(* CODESYS project CtaAppLeistungsreduktion_2.0.0.0.library
   Description: Leistungsreduktion Library der CTA
   Version: 2.0.0.0
   Title: CtaAppLeistungsreduktion
   Author: SIS
   DocFormat: reStructuredText
   LanguageModelAttribute: qualified-access-only
   Placeholder: CtaAppLeistungsreduktion
   DefaultNamespace: CtaAppLeistungsreduktion
   CompiledLibraryCompatibilityVersion: CODESYS V3.5 SP16 Patch 3
   Company: CTA

Project tree, tasks and I/O mapping:
  libraries: CtaSysConfig, 2.0.0.0 (CTA); CtaAppTime, 1.0.0.1 (CTA); CtaAppPid, 2.0.0.0 (CTA); Standard, 3.5.18.0 (System); VisuSymbols, 4.5.0.0 (System); CtaVisSymbols, 2.0.0.0 (CTA); CtaAppInfluxLog, 1.0.0.1 (CTA); VisuDialogs, * (System); CtaVisApps, 1.0.0.0 (CTA); CtaVisHelp, 1.0.0.0 (CTA); CtaVisUser, 1.0.0.0 (CTA)
  40 Visualizations/
    visualisation visLeistungsreduktion
    Powerreduction/
      Rectangles/
        visualisation visPowerReduktion4eck
        visualisation visPowerReduktion4eckCircuit
        visualisation visPowerReduktion4eckCircuitSingle
        visualisation visPowerReduktionSingle
      Combinations/
        visualisation visPrCircuit
        visualisation visPrCircuitSingle
      VisIcons/
        Circuits/
          SingleCompressor/
            visualisation visPowerReduktionKreisInOnly
            visualisation visPowerReduktionKreis
          DualCompressor/
            visualisation visPowerReduktionKreis2V
            visualisation visPowerReduktionKreis2VInOnly
        GeneralPowerreductions/
          visualisation visPrIn
          visualisation visPrInOut
          visualisation visPrOut
          visualisation visPrNoInOut
    Parameter/
      visualisation Parameter
    Dialogs/
      visualisation visLeistungsreduktionManager
      visualisation visLrZeile
  30 Program Organization Units/
    function block fbLeistungsReduktionManager [ST]
    function block fbLeistungsReduktion [ST]: actConfig, actTrendLog, actLeistungreduktion
  00000000-0000-0000-0000-000000000000|D:\CoDeSys\LibrariesV3\trunk\Intern\CAA\CAA Template\3.4.0.0 draft\Placeholder.xml
  00000000-0000-0000-0000-000000000000|D:\CoDeSys\LibrariesV3\trunk\Intern\CAA\CAA Template\3.2.0.3 draft\Prefix.pdf
  00000000-0000-0000-0000-000000000000|D:\CoDeSys\LibrariesV3\trunk\Intern\CAA\CAA Template\3.5.2.0 draft\Placeholder.xml
  20 Structs/
    data type scParameter
  50 Images/
  10 Documenation/
    global variables VersionHistory
    global variables readMe
  21 Interface/
  11 Library Parameter/
  12 Konstanten/
  60 Textlisten/
  13 Globale Variablen/
  text list GlobalTextList
*)

// 20 Structs/scParameter
TYPE scParameter :
    STRUCT
        fbxEn                         :   CtaSysConfig.fbBOOL;   // 1=Leistungsreduktion Überwachung aktivieren/deaktivieren
        fbtStartTime                  :   CtaSysConfig.fbTIME;   // Ton1= Sobald Verdichter/Anlage aktiv ist wird die Leistungsreduktion gemäss StartTime Einschaltverzögert
        fbtRunTime                    :   CtaSysConfig.fbTIME;   // Ton2= Sobald der Istwert den Sollwert überschreitet/unterschreitet wird die Leistungsreduktion minimum gemäss RunTime Einschaltverzögert unabhängig von Ton1
        fbrCounter                    :   CtaSysConfig.fbREAL;   // Soviel% wird in einer Sekunde angeglichen 0% zu PI Regler
        fbrSoll                       :   CtaSysConfig.fbREAL;   // Sollwert
        fbxEnTrendLog                 :   CtaSysConfig.fbBOOL;   // Trendlog Aktivieren       
    END_STRUCT
END_TYPE

// 10 Documenation/VersionHistory
(* 

.. image:: ../../Images/CTA_Logo.jpg
   :align: right
   :width: 15% 

**Vorlage**   


============ =========== =========== ============================================
**Date**     **Version** **Author**  **Change**
------------ ----------- ----------- --------------------------------------------
04.03.2021   0.0.0.0     SIS         Vorlage erstellt

============ =========== =========== ============================================


*)
VAR_GLOBAL
    stInfo : STRING:= '0.0.0.0, Vorlage, CTA';
END_VAR

// 10 Documenation/readMe
(*

**ReadMe**
 
|	**Empfehlung**
|
|	Die Bibliothek CtaAppLeistungredukton dient der reduktion der Leistung unter Berücksichtigung der definierten Parameter.
|	Instanzieren Sie den CtaAppLeistungredukton.fbLeistungsReduktion in ihrem Funktionsbaustein oder POU beispielsweise als fbLrx (x = Nr. der Leistungsreduktion)
|	Deklarieren Sie die Struktur Variable welche als Parameter und zur ansteuerung dienen wie im Code beispiel.
|  
| *Beispiel* 

+-----------------------+---------------------------------------------------------------------------------------------------------------------------------------------------------------------------------------------------------------------------------------------------------------------------------------------------------------------------------------------------------------------------------------------------------------------------------------+
| Beschreibung          |  Code                                                                                                                                                                                                                                                                                                                                                                                                                                 |
+=======================+=======================================================================================================================================================================================================================================================================================================================================================================================================================================+
| Pou oder SmFb         | .. code-block:: codesys                                                                                                                                                                                                                                                                                                                                                                                                               |
|                       |                                                                                                                                                                                                                                                                                                                                                                                                                                       |
|                       |	// Deklaration als VAR im POU oder dem selbsterstellten Funktionsbaustein                                                                                                                                                                                                                                                                                                                                                       	|
|                       |   VAR   																																																																																																								|
|						|	    (*Leistungsreduktionen*)																																																		 																																																|
|						|		fbLr1			: CtaAppLeistungredukton.fbLeistungsReduktion;                                                                                                                                                                                                                                                                                                                                                              	|
|						|																																																																																																										|
+-----------------------+---------------------------------------------------------------------------------------------------------------------------------------------------------------------------------------------------------------------------------------------------------------------------------------------------------------------------------------------------------------------------------------------------------------------------------------+
| Code für Init         | .. code-block:: codesys                                                                                                                                                                                                                                                                                                                                                                                                               |
|                       |   																																																																																																									|
| 						|	// Kopieren des nachfolgenden Codes in eine Action zur Initialisierung der Parameter. Zum Beispiel actConfig.																																																																														|
|                       |	{region " Stufenschaltung "}                                                                                                                                                                                                                                                                                                                                                                                                     	|
| 						|		(*Basis*)																																																																																																						|
|						|		fbLr1.scParameter.fbxEn               				(_wertInit :=	 FALSE														);		//P1 Leistungsreduktion aktiv / inaktiv																																																													|
|						|		fbLr1.scParameter.fbtStartTime						(_wertInit :=	 T#30s		, _minInit :=			, _maxInit :=			);		//P2 Einschaltverzögerung der Leistungsreduktion nach Start des Verdichters / der Analge																																																| 
|						|		fbLr1.scParameter.fbtRunTime						(_wertInit :=	 T#30s		, _minInit :=			, _maxInit :=			);		//P3 Einschaltverzögerung der Leistungsreduktion im Betrieb bei Unter- oder Überschreitung des Sollwertes																																												| 
|						|		fbLr1.scParameter.fbrCounter						(_wertInit :=		15		, _minInit :=			, _maxInit := 			);		//P4 Wert für Angleichung innert einer Sekunde																																																											| 
|						|		fbLr1.scParameter.fbrSoll							(_wertInit := 		30		, _minInit :=   		, _maxInit := 			);		//P5 Sollwert																																																																			|
|						|		fbLr1.scParameter.fbxEnTrendLog						(_wertInit := 	  TRUE														);		//P6 Aktivierung der Trendaufzeichnung 																																																													|
|						|	{endregion}                                                                                                                                                      																																																																	| 
+-----------------------+---------------------------------------------------------------------------------------------------------------------------------------------------------------------------------------------------------------------------------------------------------------------------------------------------------------------------------------------------------------------------------------------------------------------------------------+
*)                                                                                                                                                                                                                                                                                                                                                                                                                                                               
 VAR_GLOBAL                                                                                                                                                                                                                                                                                                                                                                                                                                                      
    xReadMeDone              :   BOOL;                                                                                                                                                                                                                                                                                                                                                                                                                           
END_VAR

// 30 Program Organization Units/fbLeistungsReduktionManager
FUNCTION_BLOCK fbLeistungsReduktionManager
VAR_INPUT
    rLAkt       :   REAL;
    fbLR1       :   REFERENCE TO fbLeistungsReduktion;
    fbLR2       :   REFERENCE TO fbLeistungsReduktion;
    fbLR3       :   REFERENCE TO fbLeistungsReduktion;
    fbLR4       :   REFERENCE TO fbLeistungsReduktion;
    fbLR5       :   REFERENCE TO fbLeistungsReduktion;
    fbLR6       :   REFERENCE TO fbLeistungsReduktion;
    fbLR7       :   REFERENCE TO fbLeistungsReduktion;
    fbLR8       :   REFERENCE TO fbLeistungsReduktion;    
END_VAR             
VAR_OUTPUT          
    rOut    :   REAL;
END_VAR
VAR
    ayLR          :   ARRAY[1..8] OF REAL;
    aypFbLR       :   ARRAY[1..8] OF POINTER TO fbLeistungsReduktion;
    rTemp         :   REAL;
    xNoValidRef   :   BOOL;
    iOffset       :   INT;
    iFor1         :   INT;
    iFor2         :   INT;
END_VAR

(* Array clean *)
FOR iFor1 := 1 TO 8 DO 
    ayLR[iFor1] := 0.0;
    aypFbLR[iFor1] := 0;
END_FOR;
xNoValidRef := NOT (    __ISVALIDREF(fbLR1) OR
                        __ISVALIDREF(fbLR2) OR 
                        __ISVALIDREF(fbLR3) OR
                        __ISVALIDREF(fbLR4) OR 
                        __ISVALIDREF(fbLR5) OR 
                        __ISVALIDREF(fbLR6) OR 
                        __ISVALIDREF(fbLR7) OR 
                        __ISVALIDREF(fbLR8)); 
                      
                           
(* Wert zuweisen *)
iOffset := 0;
IF __ISVALIDREF(fbLR1) THEN
    ayLR[1]     := fbLR1.rOut;
    aypFbLR[1]  := ADR( fbLR1);
ELSE 
    iOffset := iOffset + 1;    
END_IF;
IF __ISVALIDREF(fbLR2) THEN
    ayLR[2-iOffset]     := fbLR2.rOut;
    aypFbLR[2-iOffset]  := ADR( fbLR2);
ELSE 
    iOffset := iOffset + 1;    
END_IF;
IF __ISVALIDREF(fbLR3) THEN
    ayLR[3-iOffset]     := fbLR3.rOut;
    aypFbLR[3-iOffset]  := ADR( fbLR3);
ELSE 
    iOffset := iOffset + 1;  
END_IF;
IF __ISVALIDREF(fbLR4) THEN
    ayLR[4-iOffset]     := fbLR4.rOut;
    aypFbLR[4-iOffset]  := ADR( fbLR4);
ELSE 
    iOffset := iOffset + 1;  
END_IF;
IF __ISVALIDREF(fbLR5) THEN
    ayLR[5-iOffset]     := fbLR5.rOut;
    aypFbLR[5-iOffset]  := ADR( fbLR5);
ELSE 
    iOffset := iOffset + 1;  
END_IF;
IF __ISVALIDREF(fbLR6) THEN
    ayLR[6-iOffset]     := fbLR6.rOut;
    aypFbLR[6-iOffset]  := ADR( fbLR6);
ELSE 
    iOffset := iOffset + 1;  
END_IF;
IF __ISVALIDREF(fbLR7) THEN
    ayLR[7-iOffset]     := fbLR7.rOut;
    aypFbLR[7-iOffset]  := ADR( fbLR7);
ELSE 
    iOffset := iOffset + 1;  
END_IF;
IF __ISVALIDREF(fbLR8) THEN
    ayLR[8-iOffset]     := fbLR8.rOut;
    aypFbLR[8-iOffset]  := ADR(fbLR8);
ELSE 
    iOffset := iOffset + 1;  
END_IF;

(* Sortieren *)
FOR iFor1 := 1 TO 8 DO
    FOR iFor2 := 1 TO 7 DO
        IF ayLR[iFor2] < ayLR[iFor2 + 1] THEN
            rTemp           := ayLR[iFor2];
            ayLR[iFor2]     := ayLR[iFor2 + 1];     
            ayLR[iFor2 + 1] := rTemp;   
		END_IF;
	END_FOR;
END_FOR; 

(* Berechnen *)
rOut := rLAkt;
FOR iFor1 := 1 TO 8 DO 
    IF ayLR[iFor1] <> 0 THEN
        rOut := rOut - (( rOut / 100 ) * ayLR[iFor1]);
    ELSE
        EXIT;    
    END_IF;    
END_FOR;

(* Reset *)
fbLR1   REF= 0;
fbLR2   REF= 0;
fbLR3   REF= 0;
fbLR4   REF= 0;
fbLR5   REF= 0;
fbLR6   REF= 0;
fbLR7   REF= 0;
fbLR8   REF= 0;

END_FUNCTION_BLOCK

// 30 Program Organization Units/fbLeistungsReduktion
FUNCTION_BLOCK fbLeistungsReduktion
VAR_INPUT 
    stObjID                 :   STRING[25];                             // Objekt ID
    rIst                    :   REAL;                                   // Istwert
    xAct                    :   BOOL;                                   // 1=Verdichter/Anlage aktiv
    xInvert                 :   BOOL;                                   // 0=Wärme (aktiv Ist > als Soll) 1=Kälte (aktiv Ist < als Soll)
    stPhisikalischeEinheit	:   STRING[3];                              // z.B:'°C' oder 'K'  
END_VAR
VAR_OUTPUT
   rOut						:	REAL;
   xOut_LR_aktiv			:	BOOL;
END_VAR
VAR
    scParameter 			: 	scParameter;  
    fbConfigFile			:	CtaSysConfig.fbConfigFile;
	
    fbPID 					:	CtaAppPid.fbPid;
	
	fbSR					: 	SR;
	xSafetyIn				:	BOOL;
    xOutDelayStartRunn		:	BOOL;
	OutPID					:	REAL;
	SETfbSR1				:	BOOL;
	RESETSETfbSR1			:	BOOL;
	Cunter					:	REAL;
	fbSR2					:	SR;
	R_TRIG2					:	R_TRIG;
	TON1					:	Standard.TON;
	R_TRIG3					:	R_TRIG;
	fbSR3					:	SR;
	TP1						:	TP;
	TON2					:	Standard.TON;
	xEn						:	INT;
	(* Trendlog *) 
	fbTrendrValue			:	CtaAppInfluxLog.FB_LOG_NODE_REAL;

 {attribute 'instance-path'} 
 {attribute 'noinit'} 
 str: STRING;
  
END_VAR
VAR // added by the converter: edge detectors and wires of the graphical bodies
    _w1 : ANY;
    _w2, _w5 : BOOL;
    _w3, _w4 : REAL;
END_VAR

actConfig();
actLeistungreduktion();
actTrendLog();

ACTION actConfig:
fbConfigFile();

(* Parameter *)
scParameter.fbxEn               (_usiParaNr := 1, itfConfigFb := fbConfigFile); // Leistungsreduktion Aktivieren
scParameter.fbtStartTime        (_usiParaNr := 2, itfConfigFb := fbConfigFile); // Leistungsreduktion Startverzögerung
scParameter.fbtRunTime          (_usiParaNr := 3, itfConfigFb := fbConfigFile); // Leistungsreduktion Betriebsverzöerung
scParameter.fbrCounter          (_usiParaNr := 4, itfConfigFb := fbConfigFile); // Leistungsreduktion Wertangleichung
scParameter.fbrSoll             (_usiParaNr := 5, itfConfigFb := fbConfigFile); // Leistungsreduktion Sollwert
scParameter.fbxEnTrendLog       (_usiParaNr := 6, itfConfigFb := fbConfigFile); // Leistungsreduktion Trendlog Einschalten

//Parameters PID
fbPID.scParameter.fbrBand		(_WertInit :=  20.0, _MinInit := , _MaxInit :=);
fbPID.scParameter.fbrDeadBand	(_WertInit :=   0.0, _MinInit := , _MaxInit :=);
fbPID.scParameter.fbrTn			(_WertInit := 120.0, _MinInit := , _MaxInit :=);
fbPID.scParameter.fbrTv			(_WertInit :=   0.0, _MinInit := , _MaxInit :=);
fbPID.scParameter.fbxInvert		(_WertInit := FALSE);
fbPID.scParameter.fbxEnTrendlog	(_WertInit := FALSE);
END_ACTION

ACTION actTrendLog:
(* rValue *)
fbTrendrValue.ENABLE	:= 	scParameter.fbxEn.proValue 			AND
							scParameter.fbxEnTrendLog.proValue;
fbTrendrValue.KEY		:=	CONCAT(stObjID,'_rValue');
fbTrendrValue.SET_VALUE	:=	rOut;
END_ACTION

ACTION actLeistungreduktion:
TON1(IN := xAct, PT := scParameter.fbtStartTime.proValue); // Standard.TON
xOut_LR_aktiv := xOutDelayStartRunn;
TON2(IN := (SEL(xInvert, rIst > scParameter.fbrSoll.proValue, rIst < scParameter.fbrSoll.proValue) OR rOut > 0 AND xOutDelayStartRunn) AND scParameter.fbxEn.proValue, PT := scParameter.fbtRunTime.proValue); // Standard.TON
xOutDelayStartRunn := TON1.Q AND TON2.Q;
// Ton1= Sobald Verdichter/Anlage aktiv ist wird die Leistungsreduktion gemäss StartTime Einschaltverzögert
// Ton2= Sobald der Istwert den Sollwert überschreitet/unterschreitet wird die Leistungsreduktion minimum gemäss RunTime Einschaltverzögert unabhängig von Ton1
SETfbSR1 := SEL(xInvert, rIst >= scParameter.fbrSoll.proValue, rIst <= scParameter.fbrSoll.proValue) AND xOutDelayStartRunn;
fbPID.proInvert := xInvert;
fbSR2(SET1 := SETfbSR1, RESET := RESETSETfbSR1); // SR
fbPID(
    xEn := fbSR2.Q1,
    rAct := rIst,
    rSoll := scParameter.fbrSoll.proValue,
    stPhysikalischeEinheit := stPhisikalischeEinheit); // CtaAppPid.fbPid
OutPID := LIMIT(0, fbPID.rY, 100);
R_TRIG2(CLK := OutPID <= 0); // R_TRIG
RESETSETfbSR1 := R_TRIG2.Q OR NOT xAct;
IF NOT xOutDelayStartRunn THEN _w1 := 0; END_IF
Cunter := _w1;
TP1(IN := NOT TP1.Q, PT := T#1s); // TP
_w2 := xOutDelayStartRunn AND NOT TP1.Q;
IF _w2 THEN _w3 := Cunter + scParameter.fbrCounter.proValue; END_IF
IF _w2 THEN _w4 := LIMIT(0, Cunter, 102); END_IF
Cunter := _w3;
Cunter := _w4;
_w5 := xOutDelayStartRunn AND OutPID > 0;
R_TRIG3(CLK := xOutDelayStartRunn); // R_TRIG
// Da die Leistungsreduktion beim Start /Betrieb verzögert werden kann, ist es möglich das der PI Regler nach der Verzögerung bereits eine grosse Reduktion anfordert.
// Aus diesem Grund wird  über den Cunter der  Output  anlgsam angeglichen
fbSR3(SET1 := R_TRIG3.Q, RESET := Cunter >= OutPID AND xOutDelayStartRunn OR NOT xAct); // SR
rOut := SEL(_w5, 0, SEL(fbSR3.Q1, OutPID, Cunter));
END_ACTION

END_FUNCTION_BLOCK

// 40 Visualizations/visLeistungsreduktion
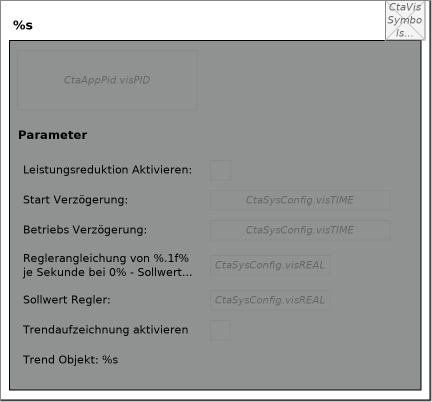
VISUALIZATION visLeistungsreduktion  // 432x402
VAR_IN_OUT
    {attribute 'VAR_IN_OUT_AS_POINTER'}
    fbLeistungsReduktion_IN  :   fbLeistungsReduktion;	
END_VAR
VAR
    iLanguage : INT;
END_VAR
    RoundedRectangle (0,0 430x400)
    RoundedRectangle (9,40 412x350)
    Image (385,0 40x40), image: CtaVisSymbols.ImagePool.close_solo_black
        OnMouseDown:  Dialog=visLeistungsreduktion, Result=None, NumpadKeypadSet=True
    Frame (17,50 180x60)
        shows CtaAppPid.visPID(fbPID := fbLeistungsReduktion_IN.fbPID)
    Textfield (10,5 400x40), "%s", text variable: fbLeistungsReduktion_IN.stObjID
    Frame (10,120 410x260)
        shows Parameter(fbLeistungsReduktion_IN := fbLeistungsReduktion_IN)
END_VISUALIZATION

// 40 Visualizations/Parameter/Parameter
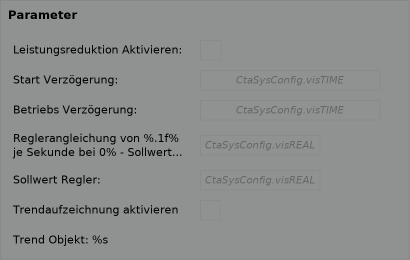
VISUALIZATION Parameter  // 410x260
VAR_IN_OUT
    fbLeistungsReduktion_IN  :   fbLeistungsReduktion;
END_VAR
    Label (5,5 150x20), "Parameter"
    Label (10,70 180x20), "Start Verzögerung:"
    Label (10,100 180x20), "Betriebs Verzögerung:"
    Frame (200,100 180x20)
        shows CtaSysConfig.visTIME(visfbTIMEIn := fbLeistungsReduktion_IN.scParameter.fbtRunTime)
    Frame (200,70 180x20)
        shows CtaSysConfig.visTIME(visfbTIMEIn := fbLeistungsReduktion_IN.scParameter.fbtStartTime)
    Label (10,40 180x20), "Leistungsreduktion Aktivieren:"
    Rectangle (10,230 395x20), "Trend Objekt: %s", text variable: fbLeistungsReduktion_IN.stObjID
    Frame (200,200 20x20)
        shows CtaSysConfig.visBOOL(visfbBOOLIn := fbLeistungsReduktion_IN.scParameter.fbxEnTrendLog)
    Label (10,200 180x20), "Trendaufzeichnung aktivieren"
    Label (10,170 180x20), "Sollwert Regler:"
    Frame (200,170 120x20)
        shows CtaSysConfig.visREAL(visfbREALIn := fbLeistungsReduktion_IN.scParameter.fbrSoll, stPhysikalischeEinheit := fbLeistungsReduktion_IN.stPhisikalischeEinheit)
    Frame (200,135 120x20)
        shows CtaSysConfig.visREAL(visfbREALIn := fbLeistungsReduktion_IN.scParameter.fbrCounter, stPhysikalischeEinheit := '%')
    Frame (200,40 21x20)
        shows CtaSysConfig.visBOOL(visfbBOOLIn := fbLeistungsReduktion_IN.scParameter.fbxEn)
    Textfield (10,130 180x30), "Reglerangleichung von %.1f% je Sekunde bei 0% - Sollwert...", text variable: fbLeistungsReduktion_IN.scParameter.fbrCounter.rValue
END_VISUALIZATION

// 40 Visualizations/Dialogs/visLeistungsreduktionManager
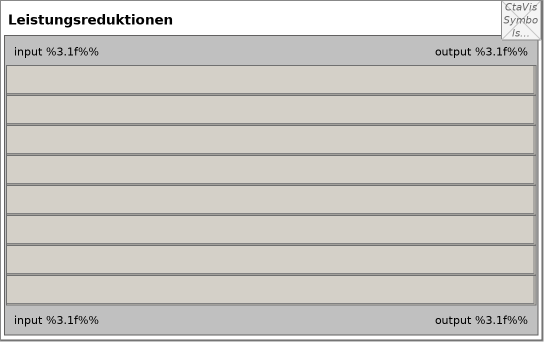
VISUALIZATION visLeistungsreduktionManager  // 544x342
VAR_IN_OUT
	{attribute 'VAR_IN_OUT_AS_POINTER'}
	fbLeistungsReduktionManager_IN : fbLeistungsReduktionManager;
END_VAR
    RoundedRectangle (0,0 542x340)
    Label (5,10 450x20), "Leistungsreduktionen"
    RoundedRectangle (4,35 534x300)
    Textfield (11,37 221x30), "input %3.1f%%", text variable: fbLeistungsReduktionManager_IN.rLAkt
    Textfield (310,37 221x30), "output %3.1f%%", text variable: fbLeistungsReduktionManager_IN.rOut
    Frame (6,65 530x30), invisible if: fbLeistungsReduktionManager_IN.aypFbLR[1] = 0
        shows visLrZeile(fbLr := fbLeistungsReduktionManager_IN.aypFbLR[1]^)
    Frame (6,95 530x30), invisible if: fbLeistungsReduktionManager_IN.aypFbLR[2] = 0
        shows visLrZeile(fbLr := fbLeistungsReduktionManager_IN.aypFbLR[2]^)
    Frame (6,125 530x30), invisible if: fbLeistungsReduktionManager_IN.aypFbLR[3] = 0
        shows visLrZeile(fbLr := fbLeistungsReduktionManager_IN.aypFbLR[3]^)
    Frame (6,155 530x30), invisible if: fbLeistungsReduktionManager_IN.aypFbLR[4] = 0
        shows visLrZeile(fbLr := fbLeistungsReduktionManager_IN.aypFbLR[4]^)
    Frame (6,185 530x30), invisible if: fbLeistungsReduktionManager_IN.aypFbLR[5] = 0
        shows visLrZeile(fbLr := fbLeistungsReduktionManager_IN.aypFbLR[5]^)
    Frame (6,215 530x30), invisible if: fbLeistungsReduktionManager_IN.aypFbLR[6] = 0
        shows visLrZeile(fbLr := fbLeistungsReduktionManager_IN.aypFbLR[6]^)
    Frame (6,245 530x30), invisible if: fbLeistungsReduktionManager_IN.aypFbLR[7] = 0
        shows visLrZeile(fbLr := fbLeistungsReduktionManager_IN.aypFbLR[7]^)
    Frame (6,275 530x30), invisible if: fbLeistungsReduktionManager_IN.aypFbLR[8] = 0
        shows visLrZeile(fbLr := fbLeistungsReduktionManager_IN.aypFbLR[8]^)
    Textfield (310,308 221x25), "output %3.1f%%", text variable: fbLeistungsReduktionManager_IN.rOut
    Textfield (11,308 221x25), "input %3.1f%%", text variable: fbLeistungsReduktionManager_IN.rLAkt
    Image (501,0 40x40), image: CtaVisSymbols.ImagePool.close_solo_black
        OnMouseDown:  Dialog=visLeistungsreduktionManager, Result=None, NumpadKeypadSet=True
END_VISUALIZATION

// 40 Visualizations/Dialogs/visLrZeile
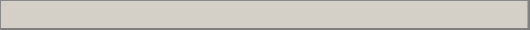
VISUALIZATION visLrZeile  // 530x30
VAR_IN_OUT
	fbLr :REFERENCE TO fbLeistungsReduktion;
END_VAR
    Textfield (0,0 250x30), "%s", text variable: fbLr.stObjID
    Textfield (250,0 80x30), "is %3.1f", text variable: fbLr.rIst
    Textfield (330,0 20x30), "%s", text variable: fbLr.stPhisikalischeEinheit
    Textfield (350,0 80x30), "set %3.1f", text variable: TO_REAL(fbLr.scParameter.fbrSoll.proValue)
    Textfield (430,0 20x30), "%s", text variable: fbLr.stPhisikalischeEinheit
    Textfield (450,0 80x30), "out %3.1f%%", text variable: fbLr.rOut
    Button (0,0 530x30)
        OnMouseClick:  Dialog=visLeistungsreduktion, Parameters={iLanguage: 1, fbLeistungsReduktion_IN: fbLr}, Selected={0: }, OpenCentered=True
END_VISUALIZATION

// 40 Visualizations/Powerreduction/Rectangles/visPowerReduktion4eck
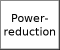
VISUALIZATION visPowerReduktion4eck  // 60x50
VAR_IN_OUT
    fbLeistungsReduktionAnlage_IN	:	fbLeistungsReduktionManager;
END_VAR
    Textfield (0,0 60x50), "Power- reduction"
        OnMouseClick:  Dialog=visLeistungsreduktionManager, Parameters={fbLeistungsReduktionManager_IN: fbLeistungsReduktionAnlage_IN}, Selected={0: }, OpenCentered=True
END_VISUALIZATION

// 40 Visualizations/Powerreduction/VisIcons/GeneralPowerreductions/visPrIn
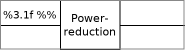
VISUALIZATION visPrIn  // 185x50
VAR_IN_OUT	
	fbLeistungsReduktionManager_IN	:	fbLeistungsReduktionManager;
END_VAR
    Rectangle (0,7 58x16), "%3.1f %%", text variable: fbLeistungsReduktionManager_IN.rLAkt
    Line (0,25) (185,25)
    Frame (60,0 60x50)
        shows visPowerReduktion4eck(fbLeistungsReduktionAnlage_IN := fbLeistungsReduktionManager_IN)
END_VISUALIZATION

// 40 Visualizations/Powerreduction/VisIcons/Circuits/SingleCompressor/visPowerReduktionKreisInOnly
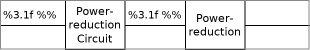
VISUALIZATION visPowerReduktionKreisInOnly  // 310x50
VAR_IN_OUT
    fbLeistungsReduktionManager_IN			: fbLeistungsReduktionManager;    
	fbLeistungsReduktionManager_IN_V1		: fbLeistungsReduktionManager;
END_VAR
    Frame (0,0 125x50)
        shows visPrCircuitSingle(fbLeistungsReduktionManager_IN := fbLeistungsReduktionManager_IN)
    Frame (125,0 185x50)
        shows visPrIn(fbLeistungsReduktionManager_IN := fbLeistungsReduktionManager_IN_V1)
END_VISUALIZATION

// 40 Visualizations/Powerreduction/VisIcons/GeneralPowerreductions/visPrInOut
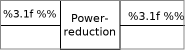
VISUALIZATION visPrInOut  // 185x50
VAR_IN_OUT	
	fbLeistungsReduktionManager_IN	:	fbLeistungsReduktionManager;
END_VAR
    Rectangle (0,5 58x18), "%3.1f %%", text variable: fbLeistungsReduktionManager_IN.rLAkt
        OnMouseClick: write the text variable via Default, min 0, max 100
    Line (0,25) (185,25)
    Rectangle (125,10 60x13), "%3.1f %%", text variable: fbLeistungsReduktionManager_IN.rOut
    Frame (60,0 60x50)
        shows visPowerReduktion4eck(fbLeistungsReduktionAnlage_IN := fbLeistungsReduktionManager_IN)
END_VISUALIZATION

// 40 Visualizations/Powerreduction/Combinations/visPrCircuit
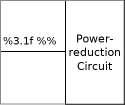
VISUALIZATION visPrCircuit  // 125x105
VAR_IN_OUT
	fbLeistungsReduktionManager_IN	:	fbLeistungsReduktionManager;
END_VAR
    Line (0,51) (119,51)
    Rectangle (0,33 58x16), "%3.1f %%", text variable: fbLeistungsReduktionManager_IN.rLAkt
        OnMouseClick: write the text variable via Default, min 0, max 100
    Frame (65,0 60x105)
        shows visPowerReduktion4eckCircuit(fbLeistungsReduktionAnlage_IN := fbLeistungsReduktionManager_IN)
END_VISUALIZATION

// 40 Visualizations/Powerreduction/Combinations/visPrCircuitSingle
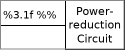
VISUALIZATION visPrCircuitSingle  // 125x50
VAR_IN_OUT
	fbLeistungsReduktionManager_IN	:	fbLeistungsReduktionManager;
END_VAR
    Line (0,25) (119,25)
    Rectangle (0,7 58x16), "%3.1f %%", text variable: fbLeistungsReduktionManager_IN.rLAkt
        OnMouseClick: write the text variable via Default, min 0, max 100
    Frame (65,0 60x50)
        shows visPowerReduktion4eckCircuitSingle(fbLeistungsReduktionAnlage_IN := fbLeistungsReduktionManager_IN)
END_VISUALIZATION

// 40 Visualizations/Powerreduction/Rectangles/visPowerReduktion4eckCircuit
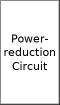
VISUALIZATION visPowerReduktion4eckCircuit  // 60x105
VAR_IN_OUT
    fbLeistungsReduktionAnlage_IN	:	fbLeistungsReduktionManager;
END_VAR
    Textfield (0,0 60x105), "Power- reduction Circuit"
        OnMouseClick:  Dialog=visLeistungsreduktionManager, Parameters={fbLeistungsReduktionManager_IN: fbLeistungsReduktionAnlage_IN}, Selected={0: }, OpenCentered=True
END_VISUALIZATION

// 40 Visualizations/Powerreduction/VisIcons/Circuits/DualCompressor/visPowerReduktionKreis2V
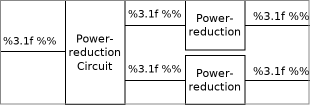
VISUALIZATION visPowerReduktionKreis2V  // 310x105
VAR_IN_OUT
    fbLeistungsReduktionManager_IN			: fbLeistungsReduktionManager;    
	fbLeistungsReduktionManager_IN_V1		: fbLeistungsReduktionManager;
    fbLeistungsReduktionManager_IN_V2		: fbLeistungsReduktionManager;
END_VAR
    Frame (0,0 125x105)
        shows visPrCircuit(fbLeistungsReduktionManager_IN := fbLeistungsReduktionManager_IN)
    Frame (125,0 185x50)
        shows visPrInOut(fbLeistungsReduktionManager_IN := fbLeistungsReduktionManager_IN_V1)
    Frame (125,55 185x50)
        shows visPrInOut(fbLeistungsReduktionManager_IN := fbLeistungsReduktionManager_IN_V2)
END_VISUALIZATION

// 40 Visualizations/Powerreduction/Rectangles/visPowerReduktion4eckCircuitSingle
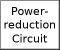
VISUALIZATION visPowerReduktion4eckCircuitSingle  // 60x50
VAR_IN_OUT
    fbLeistungsReduktionAnlage_IN	:	fbLeistungsReduktionManager;
END_VAR
    Textfield (0,0 60x50), "Power- reduction Circuit"
        OnMouseClick:  Dialog=visLeistungsreduktionManager, Parameters={fbLeistungsReduktionManager_IN: fbLeistungsReduktionAnlage_IN}, Selected={0: }, OpenCentered=True
END_VISUALIZATION

// 40 Visualizations/Powerreduction/VisIcons/GeneralPowerreductions/visPrOut
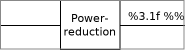
VISUALIZATION visPrOut  // 185x50
VAR_IN_OUT	
	fbLeistungsReduktionManager_IN	:	fbLeistungsReduktionManager;
END_VAR
    Line (0,25) (185,25)
    Rectangle (125,10 60x13), "%3.1f %%", text variable: fbLeistungsReduktionManager_IN.rOut
    Frame (60,0 60x50)
        shows visPowerReduktion4eck(fbLeistungsReduktionAnlage_IN := fbLeistungsReduktionManager_IN)
END_VISUALIZATION

// 40 Visualizations/Powerreduction/VisIcons/GeneralPowerreductions/visPrNoInOut
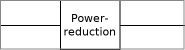
VISUALIZATION visPrNoInOut  // 185x50
VAR_IN_OUT	
	fbLeistungsReduktionManager_IN	:	fbLeistungsReduktionManager;
END_VAR
    Line (0,25) (185,25)
    Frame (60,0 60x50)
        shows visPowerReduktion4eck(fbLeistungsReduktionAnlage_IN := fbLeistungsReduktionManager_IN)
END_VISUALIZATION

// 40 Visualizations/Powerreduction/VisIcons/Circuits/SingleCompressor/visPowerReduktionKreis
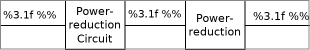
VISUALIZATION visPowerReduktionKreis  // 310x50
VAR_IN_OUT
    fbLeistungsReduktionManager_IN			: fbLeistungsReduktionManager;    
	fbLeistungsReduktionManager_IN_V1		: fbLeistungsReduktionManager;
END_VAR
    Frame (0,0 125x50)
        shows visPrCircuitSingle(fbLeistungsReduktionManager_IN := fbLeistungsReduktionManager_IN)
    Frame (125,0 185x50)
        shows visPrInOut(fbLeistungsReduktionManager_IN := fbLeistungsReduktionManager_IN_V1)
END_VISUALIZATION

// 40 Visualizations/Powerreduction/VisIcons/Circuits/DualCompressor/visPowerReduktionKreis2VInOnly
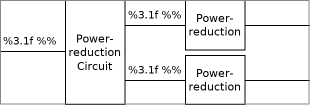
VISUALIZATION visPowerReduktionKreis2VInOnly  // 310x105
VAR_IN_OUT
    fbLeistungsReduktionManager_IN			: fbLeistungsReduktionManager;    
	fbLeistungsReduktionManager_IN_V1		: fbLeistungsReduktionManager;
    fbLeistungsReduktionManager_IN_V2		: fbLeistungsReduktionManager;
END_VAR
    Frame (0,0 125x105)
        shows visPrCircuit(fbLeistungsReduktionManager_IN := fbLeistungsReduktionManager_IN)
    Frame (125,0 185x50)
        shows visPrIn(fbLeistungsReduktionManager_IN := fbLeistungsReduktionManager_IN_V1)
    Frame (125,55 185x50)
        shows visPrIn(fbLeistungsReduktionManager_IN := fbLeistungsReduktionManager_IN_V2)
END_VISUALIZATION

// 40 Visualizations/Powerreduction/Rectangles/visPowerReduktionSingle
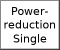
VISUALIZATION visPowerReduktionSingle  // 60x50
VAR_IN_OUT
    fbLeistungsReduktion_IN	:	fbLeistungsReduktion;
END_VAR
    Textfield (0,0 60x50), "Power- reduction Single"
        OnMouseClick:  Dialog=visLeistungsreduktion, Parameters={fbLeistungsReduktion_IN: fbLeistungsReduktion_IN, iLanguage: }, Selected={0: }, OpenCentered=True
END_VISUALIZATION
